(* Logix 5000 project; controller Ex_2_01 Emulate 5570 rev 33.11; software revision 33.00 *)
// Turn on Lamp with Push Button

TASK MainTask (continuous, watchdog 500 ms) : MainProgram

MODULES
   Local : Emulate 5570 (ICP 4, rev 33.11)
END_MODULES

VAR_GLOBAL   (* controller tags *)
   Lamp_P1 : BOOL;   // Lamp P1
   Sw_S1 : BOOL;   // Switch S1
END_VAR

PROGRAM MainProgram   (* main routine MainRoutine *)

ROUTINE MainRoutine   (* ladder *)
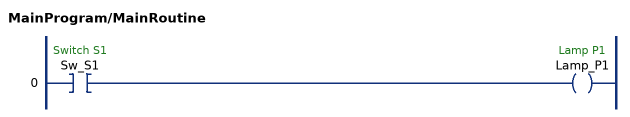
   0: XIC(Sw_S1)OTE(Lamp_P1);
END_ROUTINE
END_PROGRAM
